# EPICS substitutions: modules/SAI/SAIApp/Db/SAI_DigitalChannels.substitutions
file /opt/epics/modules/SAI/db/SAI_DigitalChannels.template {
pattern {	P,		R,		SCAN, 		ASYNPORT}
        { 	"FMB",		"MCS8:",	"1 second",	"pmac"}
}

#EOF
